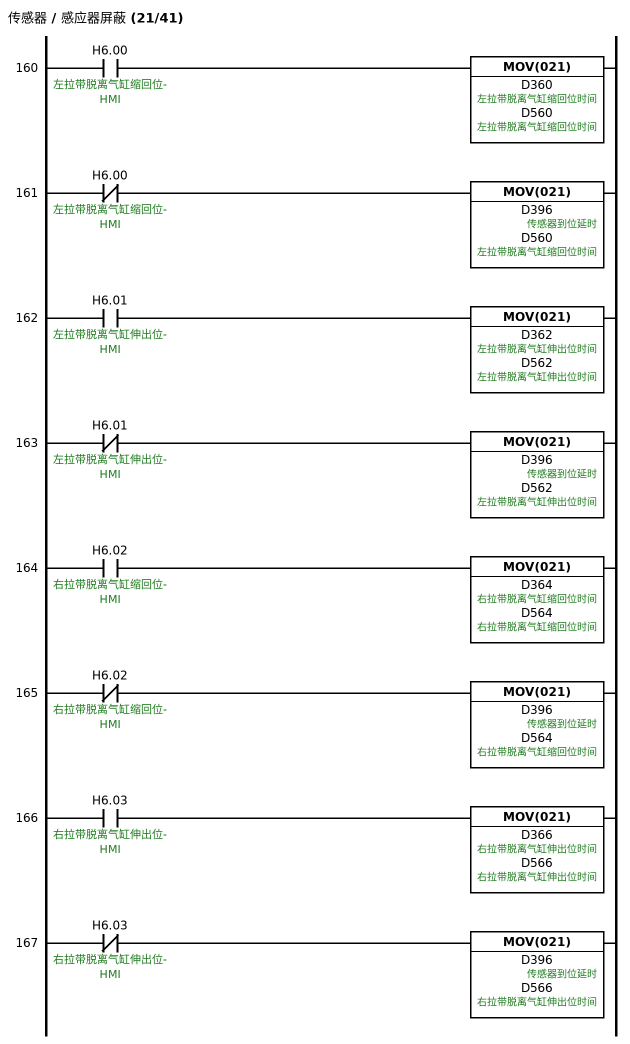
; [picture p41: 传感器 / 感应器屏蔽, rungs 160-167]
; rung 160
LD H6.00  ; 左拉带脱离气缸缩回位-HMI
MOV(021) D360 D560  ; 左拉带脱离气缸缩回位时间
; rung 161
LDNOT H6.00  ; 左拉带脱离气缸缩回位-HMI
MOV(021) D396 D560  ; 传感器到位延时, 左拉带脱离气缸缩回位时间
; rung 162
LD H6.01  ; 左拉带脱离气缸伸出位-HMI
MOV(021) D362 D562  ; 左拉带脱离气缸伸出位时间
; rung 163
LDNOT H6.01  ; 左拉带脱离气缸伸出位-HMI
MOV(021) D396 D562  ; 传感器到位延时, 左拉带脱离气缸伸出位时间
; rung 164
LD H6.02  ; 右拉带脱离气缸缩回位-HMI
MOV(021) D364 D564  ; 右拉带脱离气缸缩回位时间
; rung 165
LDNOT H6.02  ; 右拉带脱离气缸缩回位-HMI
MOV(021) D396 D564  ; 传感器到位延时, 右拉带脱离气缸缩回位时间
; rung 166
LD H6.03  ; 右拉带脱离气缸伸出位-HMI
MOV(021) D366 D566  ; 右拉带脱离气缸伸出位时间
; rung 167
LDNOT H6.03  ; 右拉带脱离气缸伸出位-HMI
MOV(021) D396 D566  ; 传感器到位延时, 右拉带脱离气缸伸出位时间

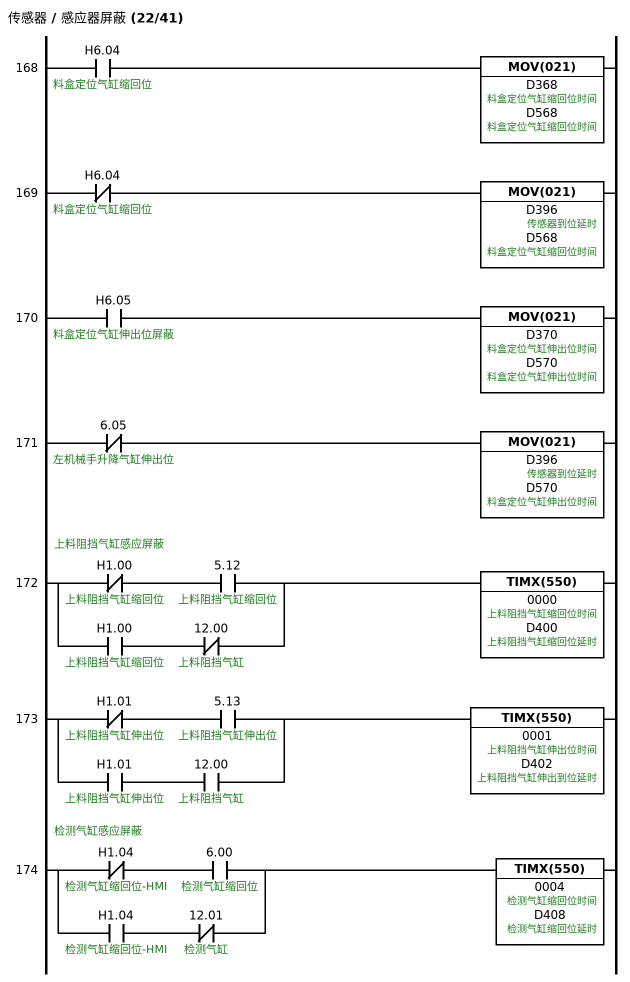
; rung 168
LD H6.04  ; 料盒定位气缸缩回位
MOV(021) D368 D568  ; 料盒定位气缸缩回位时间
; rung 169
LDNOT H6.04  ; 料盒定位气缸缩回位
MOV(021) D396 D568  ; 传感器到位延时, 料盒定位气缸缩回位时间
; rung 170
LD H6.05  ; 料盒定位气缸伸出位屏蔽
MOV(021) D370 D570  ; 料盒定位气缸伸出位时间
; rung 171
LDNOT 6.05  ; 左机械手升降气缸伸出位
MOV(021) D396 D570  ; 传感器到位延时, 料盒定位气缸伸出位时间
; rung 172: 上料阻挡气缸感应屏蔽
LDNOT H1.00  ; 上料阻挡气缸缩回位
AND 5.12  ; 上料阻挡气缸缩回位
LD H1.00  ; 上料阻挡气缸缩回位
ANDNOT 12.00  ; 上料阻挡气缸
ORLD
TIMX(550) 0000 D400  ; 上料阻挡气缸缩回位延时, 上料阻挡气缸缩回位时间
; rung 173
LDNOT H1.01  ; 上料阻挡气缸伸出位
AND 5.13  ; 上料阻挡气缸伸出位
LD H1.01  ; 上料阻挡气缸伸出位
AND 12.00  ; 上料阻挡气缸
ORLD
TIMX(550) 0001 D402  ; 上料阻挡气缸伸出到位延时, 上料阻挡气缸伸出位时间
; rung 174: 检测气缸感应屏蔽
LDNOT H1.04  ; 检测气缸缩回位-HMI
AND 6.00  ; 检测气缸缩回位
LD H1.04  ; 检测气缸缩回位-HMI
ANDNOT 12.01  ; 检测气缸
ORLD
TIMX(550) 0004 D408  ; 检测气缸缩回位延时, 检测气缸缩回位时间

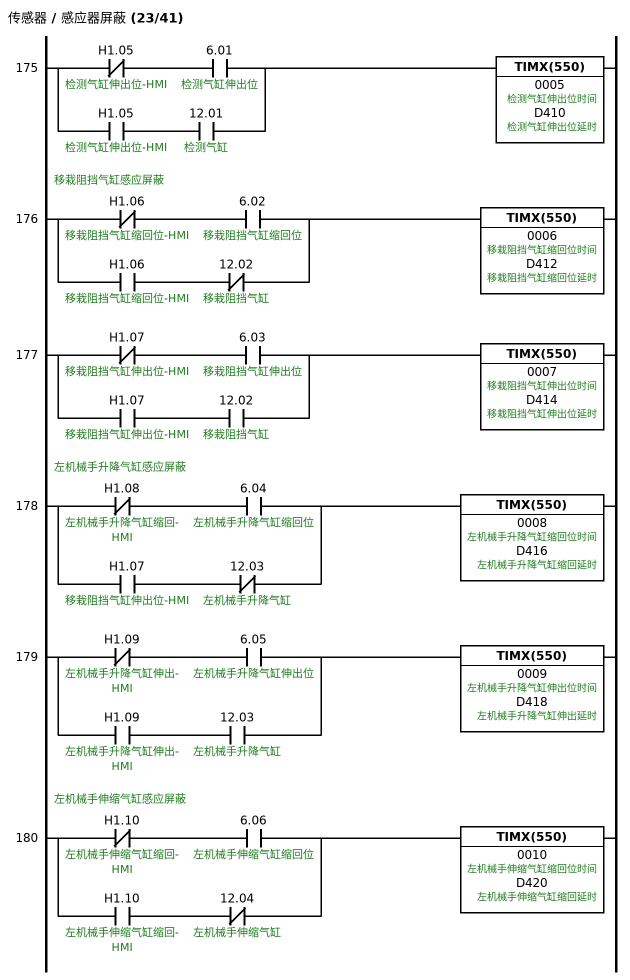
; rung 175
LDNOT H1.05  ; 检测气缸伸出位-HMI
AND 6.01  ; 检测气缸伸出位
LD H1.05  ; 检测气缸伸出位-HMI
AND 12.01  ; 检测气缸
ORLD
TIMX(550) 0005 D410  ; 检测气缸伸出位延时, 检测气缸伸出位时间
; rung 176: 移栽阻挡气缸感应屏蔽
LDNOT H1.06  ; 移栽阻挡气缸缩回位-HMI
AND 6.02  ; 移栽阻挡气缸缩回位
LD H1.06  ; 移栽阻挡气缸缩回位-HMI
ANDNOT 12.02  ; 移栽阻挡气缸
ORLD
TIMX(550) 0006 D412  ; 移栽阻挡气缸缩回位延时, 移栽阻挡气缸缩回位时间
; rung 177
LDNOT H1.07  ; 移栽阻挡气缸伸出位-HMI
AND 6.03  ; 移栽阻挡气缸伸出位
LD H1.07  ; 移栽阻挡气缸伸出位-HMI
AND 12.02  ; 移栽阻挡气缸
ORLD
TIMX(550) 0007 D414  ; 移栽阻挡气缸伸出位延时, 移栽阻挡气缸伸出位时间
; rung 178: 左机械手升降气缸感应屏蔽
LDNOT H1.08  ; 左机械手升降气缸缩回-HMI
AND 6.04  ; 左机械手升降气缸缩回位
LD H1.07  ; 移栽阻挡气缸伸出位-HMI
ANDNOT 12.03  ; 左机械手升降气缸
ORLD
TIMX(550) 0008 D416  ; 左机械手升降气缸缩回延时, 左机械手升降气缸缩回位时间
; rung 179
LDNOT H1.09  ; 左机械手升降气缸伸出-HMI
AND 6.05  ; 左机械手升降气缸伸出位
LD H1.09  ; 左机械手升降气缸伸出-HMI
AND 12.03  ; 左机械手升降气缸
ORLD
TIMX(550) 0009 D418  ; 左机械手升降气缸伸出延时, 左机械手升降气缸伸出位时间
; rung 180: 左机械手伸缩气缸感应屏蔽
LDNOT H1.10  ; 左机械手伸缩气缸缩回-HMI
AND 6.06  ; 左机械手伸缩气缸缩回位
LD H1.10  ; 左机械手伸缩气缸缩回-HMI
ANDNOT 12.04  ; 左机械手伸缩气缸
ORLD
TIMX(550) 0010 D420  ; 左机械手伸缩气缸缩回延时, 左机械手伸缩气缸缩回位时间

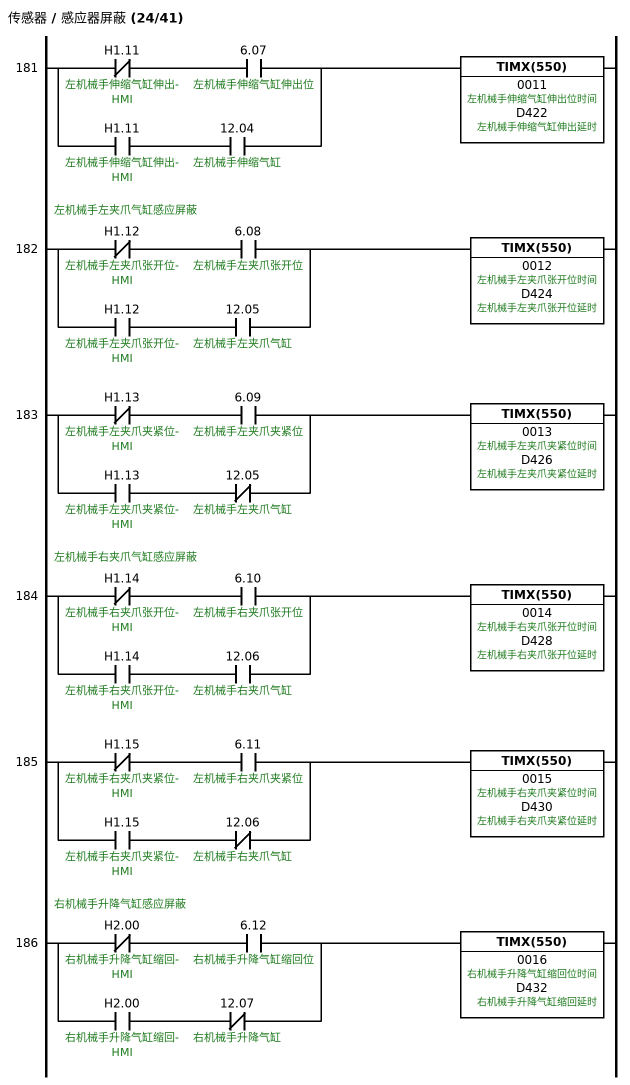
; rung 181
LDNOT H1.11  ; 左机械手伸缩气缸伸出-HMI
AND 6.07  ; 左机械手伸缩气缸伸出位
LD H1.11  ; 左机械手伸缩气缸伸出-HMI
AND 12.04  ; 左机械手伸缩气缸
ORLD
TIMX(550) 0011 D422  ; 左机械手伸缩气缸伸出延时, 左机械手伸缩气缸伸出位时间
; rung 182: 左机械手左夹爪气缸感应屏蔽
LDNOT H1.12  ; 左机械手左夹爪张开位-HMI
AND 6.08  ; 左机械手左夹爪张开位
LD H1.12  ; 左机械手左夹爪张开位-HMI
AND 12.05  ; 左机械手左夹爪气缸
ORLD
TIMX(550) 0012 D424  ; 左机械手左夹爪张开位延时, 左机械手左夹爪张开位时间
; rung 183
LDNOT H1.13  ; 左机械手左夹爪夹紧位-HMI
AND 6.09  ; 左机械手左夹爪夹紧位
LD H1.13  ; 左机械手左夹爪夹紧位-HMI
ANDNOT 12.05  ; 左机械手左夹爪气缸
ORLD
TIMX(550) 0013 D426  ; 左机械手左夹爪夹紧位延时, 左机械手左夹爪夹紧位时间
; rung 184: 左机械手右夹爪气缸感应屏蔽
LDNOT H1.14  ; 左机械手右夹爪张开位-HMI
AND 6.10  ; 左机械手右夹爪张开位
LD H1.14  ; 左机械手右夹爪张开位-HMI
AND 12.06  ; 左机械手右夹爪气缸
ORLD
TIMX(550) 0014 D428  ; 左机械手右夹爪张开位延时, 左机械手右夹爪张开位时间
; rung 185
LDNOT H1.15  ; 左机械手右夹爪夹紧位-HMI
AND 6.11  ; 左机械手右夹爪夹紧位
LD H1.15  ; 左机械手右夹爪夹紧位-HMI
ANDNOT 12.06  ; 左机械手右夹爪气缸
ORLD
TIMX(550) 0015 D430  ; 左机械手右夹爪夹紧位延时, 左机械手右夹爪夹紧位时间
; rung 186: 右机械手升降气缸感应屏蔽
LDNOT H2.00  ; 右机械手升降气缸缩回-HMI
AND 6.12  ; 右机械手升降气缸缩回位
LD H2.00  ; 右机械手升降气缸缩回-HMI
ANDNOT 12.07  ; 右机械手升降气缸
ORLD
TIMX(550) 0016 D432  ; 右机械手升降气缸缩回延时, 右机械手升降气缸缩回位时间

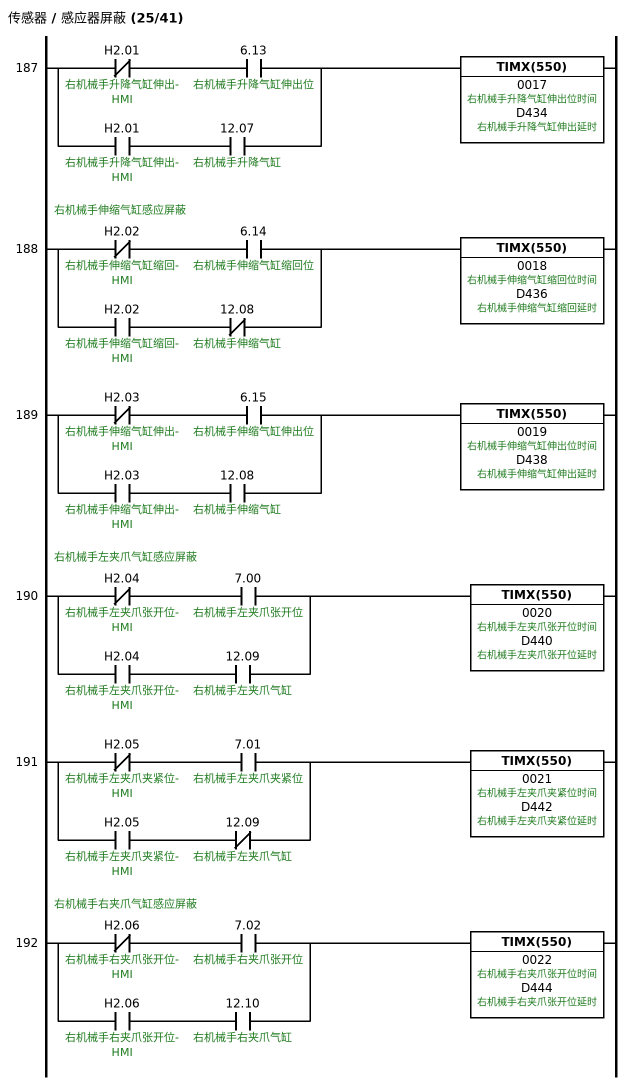
; rung 187
LDNOT H2.01  ; 右机械手升降气缸伸出-HMI
AND 6.13  ; 右机械手升降气缸伸出位
LD H2.01  ; 右机械手升降气缸伸出-HMI
AND 12.07  ; 右机械手升降气缸
ORLD
TIMX(550) 0017 D434  ; 右机械手升降气缸伸出延时, 右机械手升降气缸伸出位时间
; rung 188: 右机械手伸缩气缸感应屏蔽
LDNOT H2.02  ; 右机械手伸缩气缸缩回-HMI
AND 6.14  ; 右机械手伸缩气缸缩回位
LD H2.02  ; 右机械手伸缩气缸缩回-HMI
ANDNOT 12.08  ; 右机械手伸缩气缸
ORLD
TIMX(550) 0018 D436  ; 右机械手伸缩气缸缩回延时, 右机械手伸缩气缸缩回位时间
; rung 189
LDNOT H2.03  ; 右机械手伸缩气缸伸出-HMI
AND 6.15  ; 右机械手伸缩气缸伸出位
LD H2.03  ; 右机械手伸缩气缸伸出-HMI
AND 12.08  ; 右机械手伸缩气缸
ORLD
TIMX(550) 0019 D438  ; 右机械手伸缩气缸伸出延时, 右机械手伸缩气缸伸出位时间
; rung 190: 右机械手左夹爪气缸感应屏蔽
LDNOT H2.04  ; 右机械手左夹爪张开位-HMI
AND 7.00  ; 右机械手左夹爪张开位
LD H2.04  ; 右机械手左夹爪张开位-HMI
AND 12.09  ; 右机械手左夹爪气缸
ORLD
TIMX(550) 0020 D440  ; 右机械手左夹爪张开位延时, 右机械手左夹爪张开位时间
; rung 191
LDNOT H2.05  ; 右机械手左夹爪夹紧位-HMI
AND 7.01  ; 右机械手左夹爪夹紧位
LD H2.05  ; 右机械手左夹爪夹紧位-HMI
ANDNOT 12.09  ; 右机械手左夹爪气缸
ORLD
TIMX(550) 0021 D442  ; 右机械手左夹爪夹紧位延时, 右机械手左夹爪夹紧位时间
; rung 192: 右机械手右夹爪气缸感应屏蔽
LDNOT H2.06  ; 右机械手右夹爪张开位-HMI
AND 7.02  ; 右机械手右夹爪张开位
LD H2.06  ; 右机械手右夹爪张开位-HMI
AND 12.10  ; 右机械手右夹爪气缸
ORLD
TIMX(550) 0022 D444  ; 右机械手右夹爪张开位延时, 右机械手右夹爪张开位时间

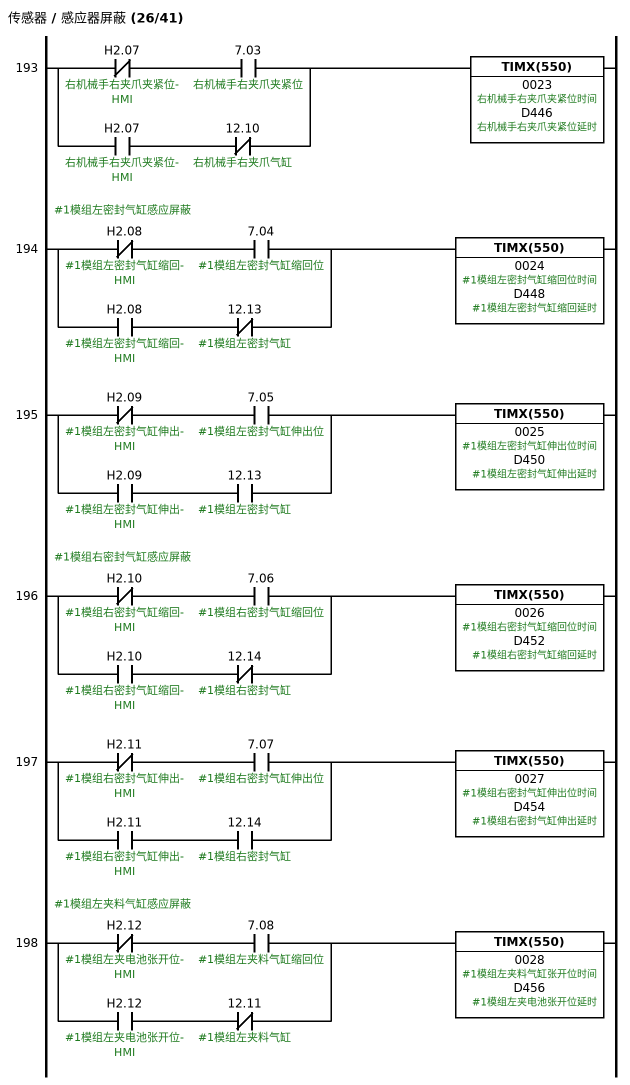
; rung 193
LDNOT H2.07  ; 右机械手右夹爪夹紧位-HMI
AND 7.03  ; 右机械手右夹爪夹紧位
LD H2.07  ; 右机械手右夹爪夹紧位-HMI
ANDNOT 12.10  ; 右机械手右夹爪气缸
ORLD
TIMX(550) 0023 D446  ; 右机械手右夹爪夹紧位延时, 右机械手右夹爪夹紧位时间
; rung 194: #1模组左密封气缸感应屏蔽
LDNOT H2.08  ; #1模组左密封气缸缩回-HMI
AND 7.04  ; #1模组左密封气缸缩回位
LD H2.08  ; #1模组左密封气缸缩回-HMI
ANDNOT 12.13  ; #1模组左密封气缸
ORLD
TIMX(550) 0024 D448  ; #1模组左密封气缸缩回延时, #1模组左密封气缸缩回位时间
; rung 195
LDNOT H2.09  ; #1模组左密封气缸伸出-HMI
AND 7.05  ; #1模组左密封气缸伸出位
LD H2.09  ; #1模组左密封气缸伸出-HMI
AND 12.13  ; #1模组左密封气缸
ORLD
TIMX(550) 0025 D450  ; #1模组左密封气缸伸出延时, #1模组左密封气缸伸出位时间
; rung 196: #1模组右密封气缸感应屏蔽
LDNOT H2.10  ; #1模组右密封气缸缩回-HMI
AND 7.06  ; #1模组右密封气缸缩回位
LD H2.10  ; #1模组右密封气缸缩回-HMI
ANDNOT 12.14  ; #1模组右密封气缸
ORLD
TIMX(550) 0026 D452  ; #1模组右密封气缸缩回延时, #1模组右密封气缸缩回位时间
; rung 197
LDNOT H2.11  ; #1模组右密封气缸伸出-HMI
AND 7.07  ; #1模组右密封气缸伸出位
LD H2.11  ; #1模组右密封气缸伸出-HMI
AND 12.14  ; #1模组右密封气缸
ORLD
TIMX(550) 0027 D454  ; #1模组右密封气缸伸出延时, #1模组右密封气缸伸出位时间
; rung 198: #1模组左夹料气缸感应屏蔽
LDNOT H2.12  ; #1模组左夹电池张开位-HMI
AND 7.08  ; #1模组左夹料气缸缩回位
LD H2.12  ; #1模组左夹电池张开位-HMI
ANDNOT 12.11  ; #1模组左夹料气缸
ORLD
TIMX(550) 0028 D456  ; #1模组左夹电池张开位延时, #1模组左夹料气缸张开位时间

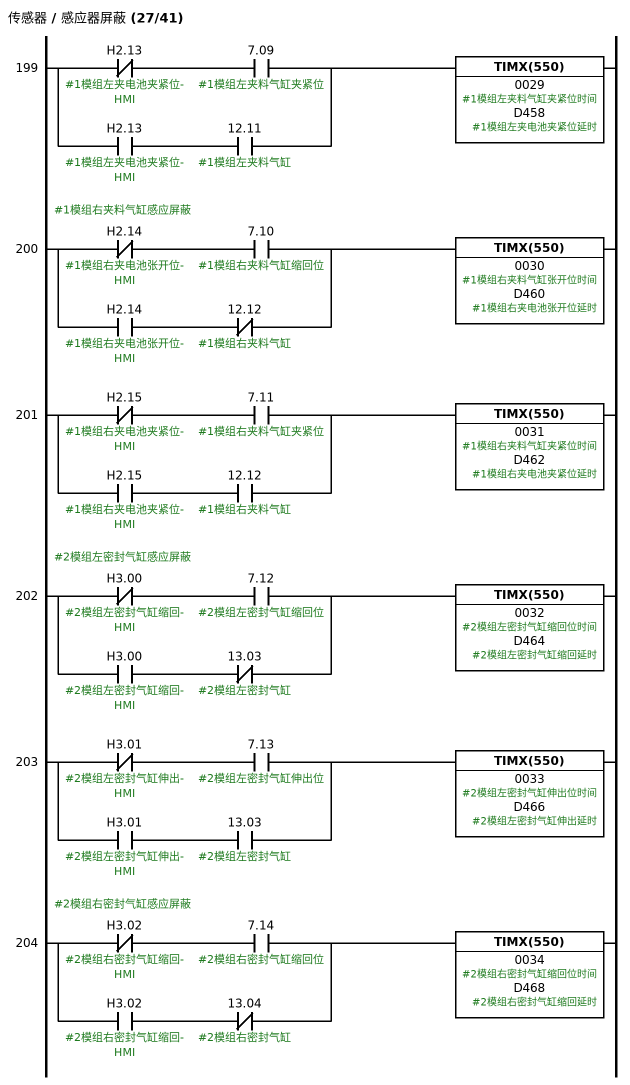
; rung 199
LDNOT H2.13  ; #1模组左夹电池夹紧位-HMI
AND 7.09  ; #1模组左夹料气缸夹紧位
LD H2.13  ; #1模组左夹电池夹紧位-HMI
AND 12.11  ; #1模组左夹料气缸
ORLD
TIMX(550) 0029 D458  ; #1模组左夹电池夹紧位延时, #1模组左夹料气缸夹紧位时间
; rung 200: #1模组右夹料气缸感应屏蔽
LDNOT H2.14  ; #1模组右夹电池张开位-HMI
AND 7.10  ; #1模组右夹料气缸缩回位
LD H2.14  ; #1模组右夹电池张开位-HMI
ANDNOT 12.12  ; #1模组右夹料气缸
ORLD
TIMX(550) 0030 D460  ; #1模组右夹电池张开位延时, #1模组右夹料气缸张开位时间
; rung 201
LDNOT H2.15  ; #1模组右夹电池夹紧位-HMI
AND 7.11  ; #1模组右夹料气缸夹紧位
LD H2.15  ; #1模组右夹电池夹紧位-HMI
AND 12.12  ; #1模组右夹料气缸
ORLD
TIMX(550) 0031 D462  ; #1模组右夹电池夹紧位延时, #1模组右夹料气缸夹紧位时间
; rung 202: #2模组左密封气缸感应屏蔽
LDNOT H3.00  ; #2模组左密封气缸缩回-HMI
AND 7.12  ; #2模组左密封气缸缩回位
LD H3.00  ; #2模组左密封气缸缩回-HMI
ANDNOT 13.03  ; #2模组左密封气缸
ORLD
TIMX(550) 0032 D464  ; #2模组左密封气缸缩回延时, #2模组左密封气缸缩回位时间
; rung 203
LDNOT H3.01  ; #2模组左密封气缸伸出-HMI
AND 7.13  ; #2模组左密封气缸伸出位
LD H3.01  ; #2模组左密封气缸伸出-HMI
AND 13.03  ; #2模组左密封气缸
ORLD
TIMX(550) 0033 D466  ; #2模组左密封气缸伸出延时, #2模组左密封气缸伸出位时间
; rung 204: #2模组右密封气缸感应屏蔽
LDNOT H3.02  ; #2模组右密封气缸缩回-HMI
AND 7.14  ; #2模组右密封气缸缩回位
LD H3.02  ; #2模组右密封气缸缩回-HMI
ANDNOT 13.04  ; #2模组右密封气缸
ORLD
TIMX(550) 0034 D468  ; #2模组右密封气缸缩回延时, #2模组右密封气缸缩回位时间

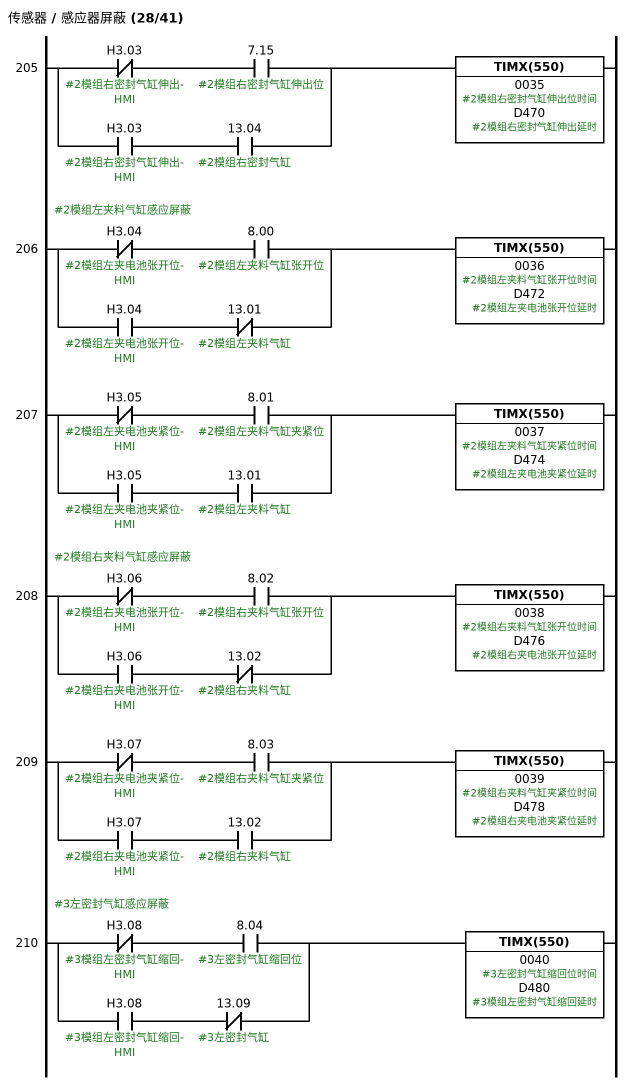
; rung 205
LDNOT H3.03  ; #2模组右密封气缸伸出-HMI
AND 7.15  ; #2模组右密封气缸伸出位
LD H3.03  ; #2模组右密封气缸伸出-HMI
AND 13.04  ; #2模组右密封气缸
ORLD
TIMX(550) 0035 D470  ; #2模组右密封气缸伸出延时, #2模组右密封气缸伸出位时间
; rung 206: #2模组左夹料气缸感应屏蔽
LDNOT H3.04  ; #2模组左夹电池张开位-HMI
AND 8.00  ; #2模组左夹料气缸张开位
LD H3.04  ; #2模组左夹电池张开位-HMI
ANDNOT 13.01  ; #2模组左夹料气缸
ORLD
TIMX(550) 0036 D472  ; #2模组左夹电池张开位延时, #2模组左夹料气缸张开位时间
; rung 207
LDNOT H3.05  ; #2模组左夹电池夹紧位-HMI
AND 8.01  ; #2模组左夹料气缸夹紧位
LD H3.05  ; #2模组左夹电池夹紧位-HMI
AND 13.01  ; #2模组左夹料气缸
ORLD
TIMX(550) 0037 D474  ; #2模组左夹电池夹紧位延时, #2模组左夹料气缸夹紧位时间
; rung 208: #2模组右夹料气缸感应屏蔽
LDNOT H3.06  ; #2模组右夹电池张开位-HMI
AND 8.02  ; #2模组右夹料气缸张开位
LD H3.06  ; #2模组右夹电池张开位-HMI
ANDNOT 13.02  ; #2模组右夹料气缸
ORLD
TIMX(550) 0038 D476  ; #2模组右夹电池张开位延时, #2模组右夹料气缸张开位时间
; rung 209
LDNOT H3.07  ; #2模组右夹电池夹紧位-HMI
AND 8.03  ; #2模组右夹料气缸夹紧位
LD H3.07  ; #2模组右夹电池夹紧位-HMI
AND 13.02  ; #2模组右夹料气缸
ORLD
TIMX(550) 0039 D478  ; #2模组右夹电池夹紧位延时, #2模组右夹料气缸夹紧位时间
; rung 210: #3左密封气缸感应屏蔽
LDNOT H3.08  ; #3模组左密封气缸缩回-HMI
AND 8.04  ; #3左密封气缸缩回位
LD H3.08  ; #3模组左密封气缸缩回-HMI
ANDNOT 13.09  ; #3左密封气缸
ORLD
TIMX(550) 0040 D480  ; #3模组左密封气缸缩回延时, #3左密封气缸缩回位时间

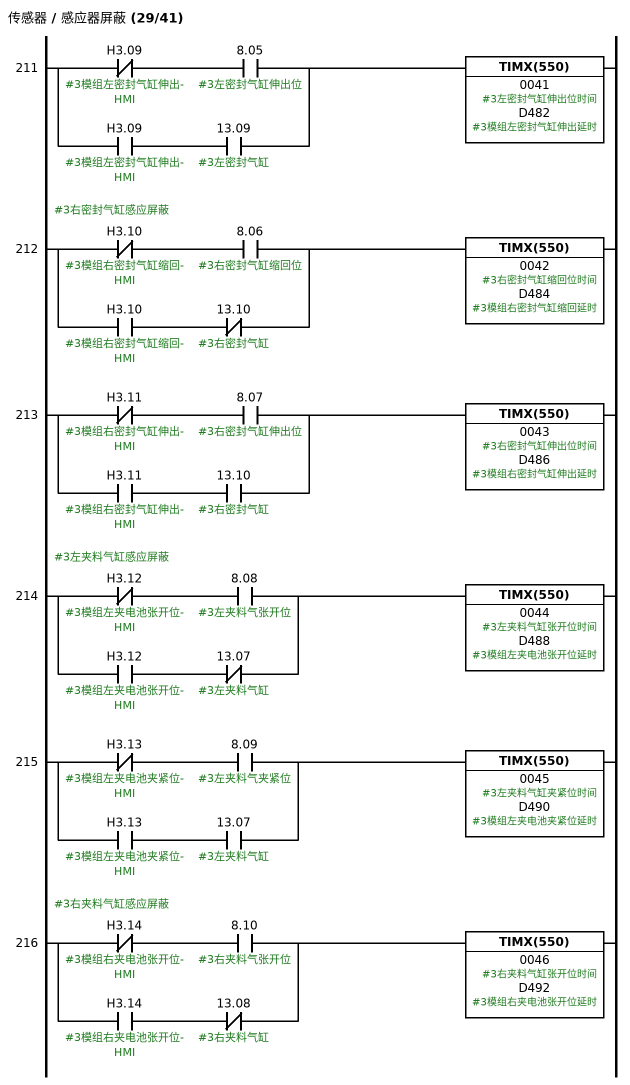
; rung 211
LDNOT H3.09  ; #3模组左密封气缸伸出-HMI
AND 8.05  ; #3左密封气缸伸出位
LD H3.09  ; #3模组左密封气缸伸出-HMI
AND 13.09  ; #3左密封气缸
ORLD
TIMX(550) 0041 D482  ; #3模组左密封气缸伸出延时, #3左密封气缸伸出位时间
; rung 212: #3右密封气缸感应屏蔽
LDNOT H3.10  ; #3模组右密封气缸缩回-HMI
AND 8.06  ; #3右密封气缸缩回位
LD H3.10  ; #3模组右密封气缸缩回-HMI
ANDNOT 13.10  ; #3右密封气缸
ORLD
TIMX(550) 0042 D484  ; #3模组右密封气缸缩回延时, #3右密封气缸缩回位时间
; rung 213
LDNOT H3.11  ; #3模组右密封气缸伸出-HMI
AND 8.07  ; #3右密封气缸伸出位
LD H3.11  ; #3模组右密封气缸伸出-HMI
AND 13.10  ; #3右密封气缸
ORLD
TIMX(550) 0043 D486  ; #3模组右密封气缸伸出延时, #3右密封气缸伸出位时间
; rung 214: #3左夹料气缸感应屏蔽
LDNOT H3.12  ; #3模组左夹电池张开位-HMI
AND 8.08  ; #3左夹料气张开位
LD H3.12  ; #3模组左夹电池张开位-HMI
ANDNOT 13.07  ; #3左夹料气缸
ORLD
TIMX(550) 0044 D488  ; #3模组左夹电池张开位延时, #3左夹料气缸张开位时间
; rung 215
LDNOT H3.13  ; #3模组左夹电池夹紧位-HMI
AND 8.09  ; #3左夹料气夹紧位
LD H3.13  ; #3模组左夹电池夹紧位-HMI
AND 13.07  ; #3左夹料气缸
ORLD
TIMX(550) 0045 D490  ; #3模组左夹电池夹紧位延时, #3左夹料气缸夹紧位时间
; rung 216: #3右夹料气缸感应屏蔽
LDNOT H3.14  ; #3模组右夹电池张开位-HMI
AND 8.10  ; #3右夹料气张开位
LD H3.14  ; #3模组右夹电池张开位-HMI
ANDNOT 13.08  ; #3右夹料气缸
ORLD
TIMX(550) 0046 D492  ; #3模组右夹电池张开位延时, #3右夹料气缸张开位时间

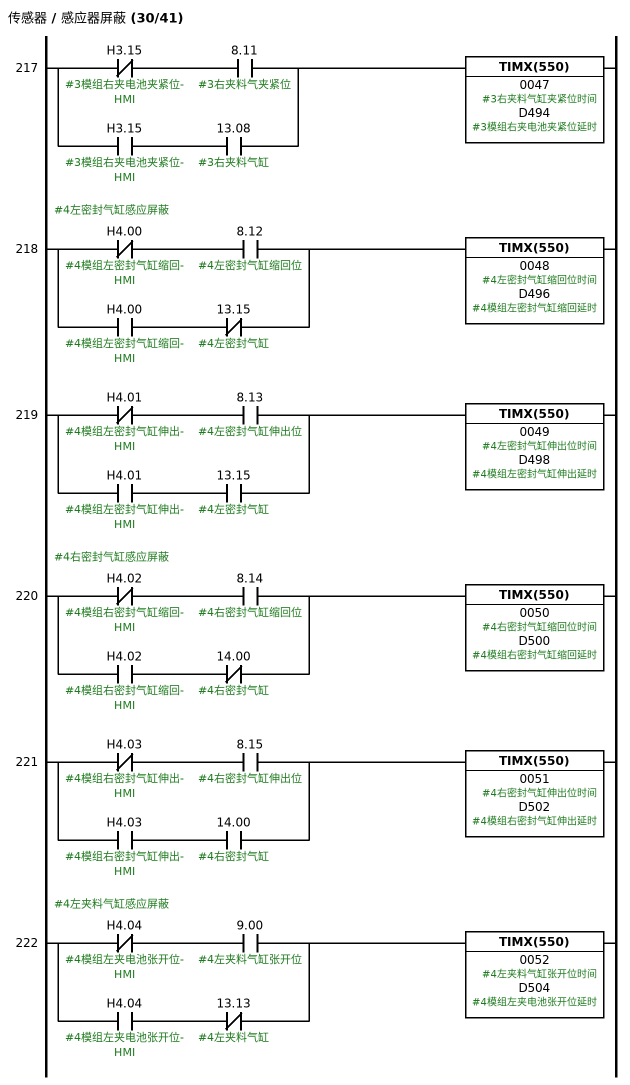
; rung 217
LDNOT H3.15  ; #3模组右夹电池夹紧位-HMI
AND 8.11  ; #3右夹料气夹紧位
LD H3.15  ; #3模组右夹电池夹紧位-HMI
AND 13.08  ; #3右夹料气缸
ORLD
TIMX(550) 0047 D494  ; #3模组右夹电池夹紧位延时, #3右夹料气缸夹紧位时间
; rung 218: #4左密封气缸感应屏蔽
LDNOT H4.00  ; #4模组左密封气缸缩回-HMI
AND 8.12  ; #4左密封气缸缩回位
LD H4.00  ; #4模组左密封气缸缩回-HMI
ANDNOT 13.15  ; #4左密封气缸
ORLD
TIMX(550) 0048 D496  ; #4模组左密封气缸缩回延时, #4左密封气缸缩回位时间
; rung 219
LDNOT H4.01  ; #4模组左密封气缸伸出-HMI
AND 8.13  ; #4左密封气缸伸出位
LD H4.01  ; #4模组左密封气缸伸出-HMI
AND 13.15  ; #4左密封气缸
ORLD
TIMX(550) 0049 D498  ; #4模组左密封气缸伸出延时, #4左密封气缸伸出位时间
; rung 220: #4右密封气缸感应屏蔽
LDNOT H4.02  ; #4模组右密封气缸缩回-HMI
AND 8.14  ; #4右密封气缸缩回位
LD H4.02  ; #4模组右密封气缸缩回-HMI
ANDNOT 14.00  ; #4右密封气缸
ORLD
TIMX(550) 0050 D500  ; #4模组右密封气缸缩回延时, #4右密封气缸缩回位时间
; rung 221
LDNOT H4.03  ; #4模组右密封气缸伸出-HMI
AND 8.15  ; #4右密封气缸伸出位
LD H4.03  ; #4模组右密封气缸伸出-HMI
AND 14.00  ; #4右密封气缸
ORLD
TIMX(550) 0051 D502  ; #4模组右密封气缸伸出延时, #4右密封气缸伸出位时间
; rung 222: #4左夹料气缸感应屏蔽
LDNOT H4.04  ; #4模组左夹电池张开位-HMI
AND 9.00  ; #4左夹料气缸张开位
LD H4.04  ; #4模组左夹电池张开位-HMI
ANDNOT 13.13  ; #4左夹料气缸
ORLD
TIMX(550) 0052 D504  ; #4模组左夹电池张开位延时, #4左夹料气缸张开位时间

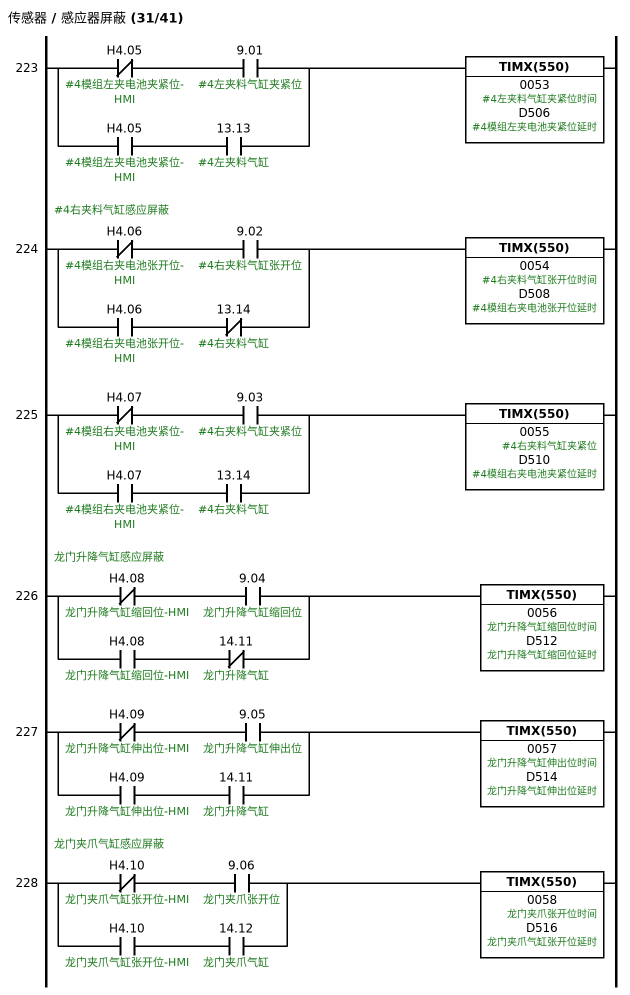
; rung 223
LDNOT H4.05  ; #4模组左夹电池夹紧位-HMI
AND 9.01  ; #4左夹料气缸夹紧位
LD H4.05  ; #4模组左夹电池夹紧位-HMI
AND 13.13  ; #4左夹料气缸
ORLD
TIMX(550) 0053 D506  ; #4模组左夹电池夹紧位延时, #4左夹料气缸夹紧位时间
; rung 224: #4右夹料气缸感应屏蔽
LDNOT H4.06  ; #4模组右夹电池张开位-HMI
AND 9.02  ; #4右夹料气缸张开位
LD H4.06  ; #4模组右夹电池张开位-HMI
ANDNOT 13.14  ; #4右夹料气缸
ORLD
TIMX(550) 0054 D508  ; #4模组右夹电池张开位延时, #4右夹料气缸张开位时间
; rung 225
LDNOT H4.07  ; #4模组右夹电池夹紧位-HMI
AND 9.03  ; #4右夹料气缸夹紧位
LD H4.07  ; #4模组右夹电池夹紧位-HMI
AND 13.14  ; #4右夹料气缸
ORLD
TIMX(550) 0055 D510  ; #4模组右夹电池夹紧位延时, #4右夹料气缸夹紧位
; rung 226: 龙门升降气缸感应屏蔽
LDNOT H4.08  ; 龙门升降气缸缩回位-HMI
AND 9.04  ; 龙门升降气缸缩回位
LD H4.08  ; 龙门升降气缸缩回位-HMI
ANDNOT 14.11  ; 龙门升降气缸
ORLD
TIMX(550) 0056 D512  ; 龙门升降气缸缩回位延时, 龙门升降气缸缩回位时间
; rung 227
LDNOT H4.09  ; 龙门升降气缸伸出位-HMI
AND 9.05  ; 龙门升降气缸伸出位
LD H4.09  ; 龙门升降气缸伸出位-HMI
AND 14.11  ; 龙门升降气缸
ORLD
TIMX(550) 0057 D514  ; 龙门升降气缸伸出位延时, 龙门升降气缸伸出位时间
; rung 228: 龙门夹爪气缸感应屏蔽
LDNOT H4.10  ; 龙门夹爪气缸张开位-HMI
AND 9.06  ; 龙门夹爪张开位
LD H4.10  ; 龙门夹爪气缸张开位-HMI
AND 14.12  ; 龙门夹爪气缸
ORLD
TIMX(550) 0058 D516  ; 龙门夹爪气缸张开位延时, 龙门夹爪张开位时间

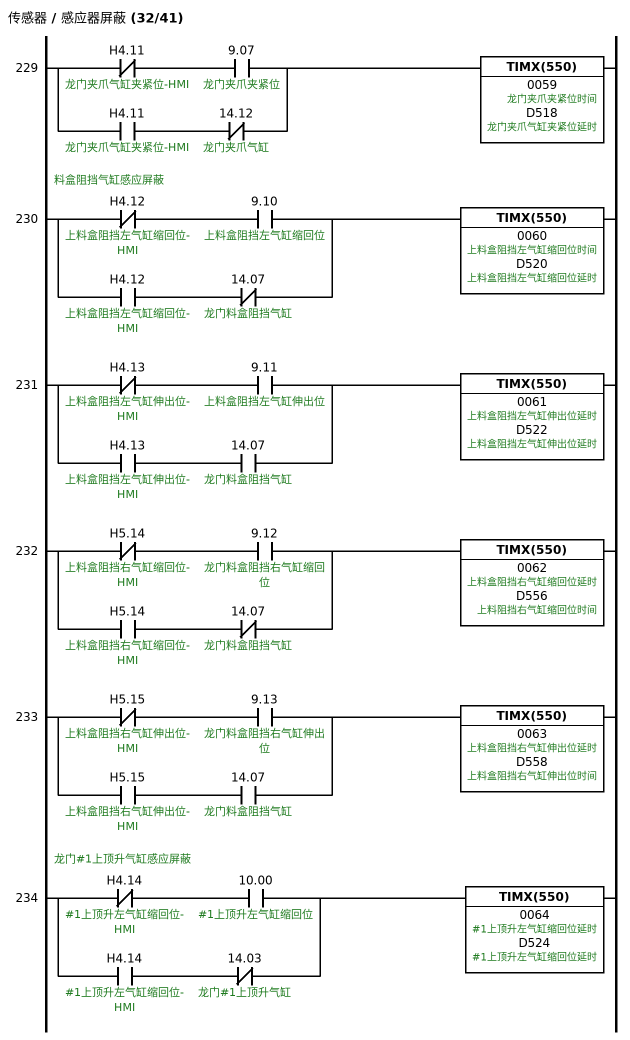
; rung 229
LDNOT H4.11  ; 龙门夹爪气缸夹紧位-HMI
AND 9.07  ; 龙门夹爪夹紧位
LD H4.11  ; 龙门夹爪气缸夹紧位-HMI
ANDNOT 14.12  ; 龙门夹爪气缸
ORLD
TIMX(550) 0059 D518  ; 龙门夹爪气缸夹紧位延时, 龙门夹爪夹紧位时间
; rung 230: 料盒阻挡气缸感应屏蔽
LDNOT H4.12  ; 上料盒阻挡左气缸缩回位-HMI
AND 9.10  ; 上料盒阻挡左气缸缩回位
LD H4.12  ; 上料盒阻挡左气缸缩回位-HMI
ANDNOT 14.07  ; 龙门料盒阻挡气缸
ORLD
TIMX(550) 0060 D520  ; 上料盒阻挡左气缸缩回位延时, 上料盒阻挡左气缸缩回位时间
; rung 231
LDNOT H4.13  ; 上料盒阻挡左气缸伸出位-HMI
AND 9.11  ; 上料盒阻挡左气缸伸出位
LD H4.13  ; 上料盒阻挡左气缸伸出位-HMI
AND 14.07  ; 龙门料盒阻挡气缸
ORLD
TIMX(550) 0061 D522  ; 上料盒阻挡左气缸伸出位延时
; rung 232
LDNOT H5.14  ; 上料盒阻挡右气缸缩回位-HMI
AND 9.12  ; 龙门料盒阻挡右气缸缩回位
LD H5.14  ; 上料盒阻挡右气缸缩回位-HMI
ANDNOT 14.07  ; 龙门料盒阻挡气缸
ORLD
TIMX(550) 0062 D556  ; 上料阻挡右气缸缩回位时间, 上料盒阻挡右气缸缩回位延时
; rung 233
LDNOT H5.15  ; 上料盒阻挡右气缸伸出位-HMI
AND 9.13  ; 龙门料盒阻挡右气缸伸出位
LD H5.15  ; 上料盒阻挡右气缸伸出位-HMI
AND 14.07  ; 龙门料盒阻挡气缸
ORLD
TIMX(550) 0063 D558  ; 上料盒阻挡右气缸伸出位时间, 上料盒阻挡右气缸伸出位延时
; rung 234: 龙门#1上顶升气缸感应屏蔽
LDNOT H4.14  ; #1上顶升左气缸缩回位-HMI
AND 10.00  ; #1上顶升左气缸缩回位
LD H4.14  ; #1上顶升左气缸缩回位-HMI
ANDNOT 14.03  ; 龙门#1上顶升气缸
ORLD
TIMX(550) 0064 D524  ; #1上顶升左气缸缩回位延时

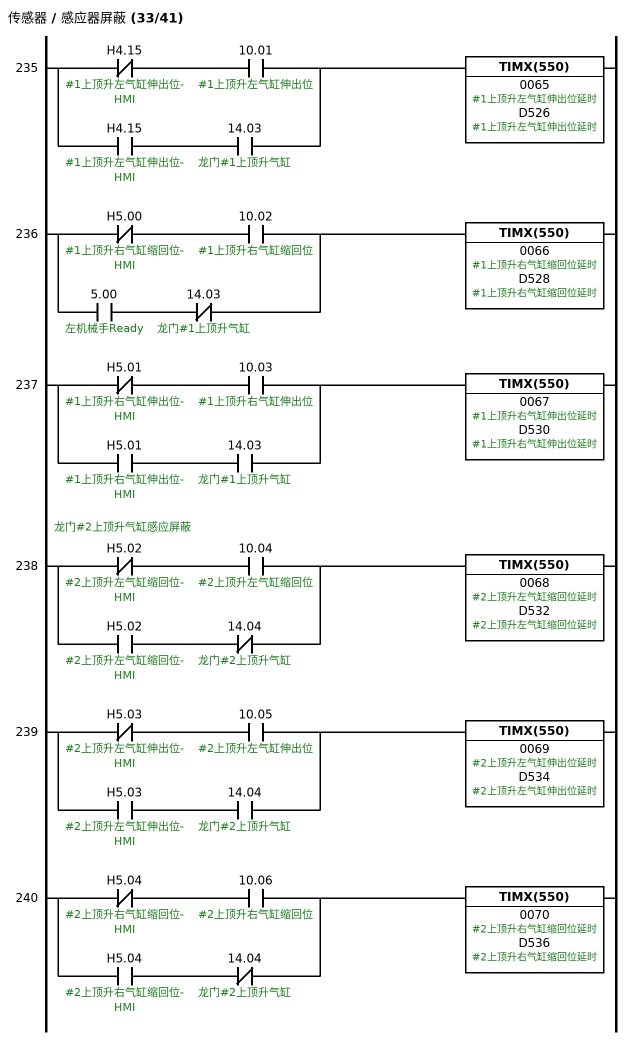
; rung 235
LDNOT H4.15  ; #1上顶升左气缸伸出位-HMI
AND 10.01  ; #1上顶升左气缸伸出位
LD H4.15  ; #1上顶升左气缸伸出位-HMI
AND 14.03  ; 龙门#1上顶升气缸
ORLD
TIMX(550) 0065 D526  ; #1上顶升左气缸伸出位延时
; rung 236
LDNOT H5.00  ; #1上顶升右气缸缩回位-HMI
AND 10.02  ; #1上顶升右气缸缩回位
LD 5.00  ; 左机械手Ready
ANDNOT 14.03  ; 龙门#1上顶升气缸
ORLD
TIMX(550) 0066 D528  ; #1上顶升右气缸缩回位延时
; rung 237
LDNOT H5.01  ; #1上顶升右气缸伸出位-HMI
AND 10.03  ; #1上顶升右气缸伸出位
LD H5.01  ; #1上顶升右气缸伸出位-HMI
AND 14.03  ; 龙门#1上顶升气缸
ORLD
TIMX(550) 0067 D530  ; #1上顶升右气缸伸出位延时
; rung 238: 龙门#2上顶升气缸感应屏蔽
LDNOT H5.02  ; #2上顶升左气缸缩回位-HMI
AND 10.04  ; #2上顶升左气缸缩回位
LD H5.02  ; #2上顶升左气缸缩回位-HMI
ANDNOT 14.04  ; 龙门#2上顶升气缸
ORLD
TIMX(550) 0068 D532  ; #2上顶升左气缸缩回位延时
; rung 239
LDNOT H5.03  ; #2上顶升左气缸伸出位-HMI
AND 10.05  ; #2上顶升左气缸伸出位
LD H5.03  ; #2上顶升左气缸伸出位-HMI
AND 14.04  ; 龙门#2上顶升气缸
ORLD
TIMX(550) 0069 D534  ; #2上顶升左气缸伸出位延时
; rung 240
LDNOT H5.04  ; #2上顶升右气缸缩回位-HMI
AND 10.06  ; #2上顶升右气缸缩回位
LD H5.04  ; #2上顶升右气缸缩回位-HMI
ANDNOT 14.04  ; 龙门#2上顶升气缸
ORLD
TIMX(550) 0070 D536  ; #2上顶升右气缸缩回位延时

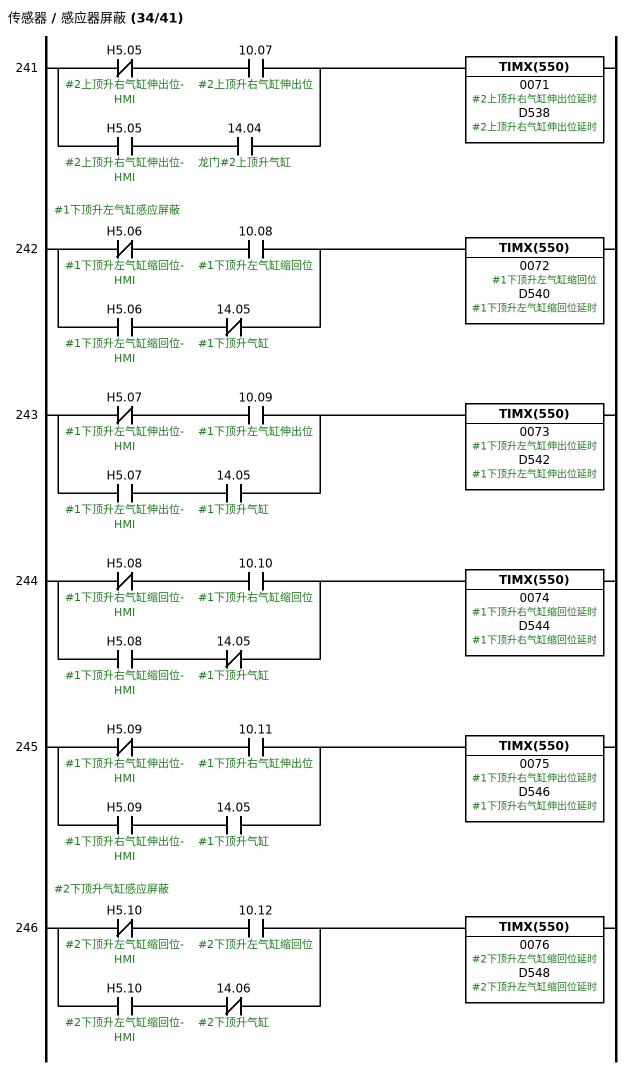
; rung 241
LDNOT H5.05  ; #2上顶升右气缸伸出位-HMI
AND 10.07  ; #2上顶升右气缸伸出位
LD H5.05  ; #2上顶升右气缸伸出位-HMI
AND 14.04  ; 龙门#2上顶升气缸
ORLD
TIMX(550) 0071 D538  ; #2上顶升右气缸伸出位延时
; rung 242: #1下顶升左气缸感应屏蔽
LDNOT H5.06  ; #1下顶升左气缸缩回位-HMI
AND 10.08  ; #1下顶升左气缸缩回位
LD H5.06  ; #1下顶升左气缸缩回位-HMI
ANDNOT 14.05  ; #1下顶升气缸
ORLD
TIMX(550) 0072 D540  ; #1下顶升左气缸缩回位延时, #1下顶升左气缸缩回位
; rung 243
LDNOT H5.07  ; #1下顶升左气缸伸出位-HMI
AND 10.09  ; #1下顶升左气缸伸出位
LD H5.07  ; #1下顶升左气缸伸出位-HMI
AND 14.05  ; #1下顶升气缸
ORLD
TIMX(550) 0073 D542  ; #1下顶升左气缸伸出位延时
; rung 244
LDNOT H5.08  ; #1下顶升右气缸缩回位-HMI
AND 10.10  ; #1下顶升右气缸缩回位
LD H5.08  ; #1下顶升右气缸缩回位-HMI
ANDNOT 14.05  ; #1下顶升气缸
ORLD
TIMX(550) 0074 D544  ; #1下顶升右气缸缩回位延时
; rung 245
LDNOT H5.09  ; #1下顶升右气缸伸出位-HMI
AND 10.11  ; #1下顶升右气缸伸出位
LD H5.09  ; #1下顶升右气缸伸出位-HMI
AND 14.05  ; #1下顶升气缸
ORLD
TIMX(550) 0075 D546  ; #1下顶升右气缸伸出位延时
; rung 246: #2下顶升气缸感应屏蔽
LDNOT H5.10  ; #2下顶升左气缸缩回位-HMI
AND 10.12  ; #2下顶升左气缸缩回位
LD H5.10  ; #2下顶升左气缸缩回位-HMI
ANDNOT 14.06  ; #2下顶升气缸
ORLD
TIMX(550) 0076 D548  ; #2下顶升左气缸缩回位延时

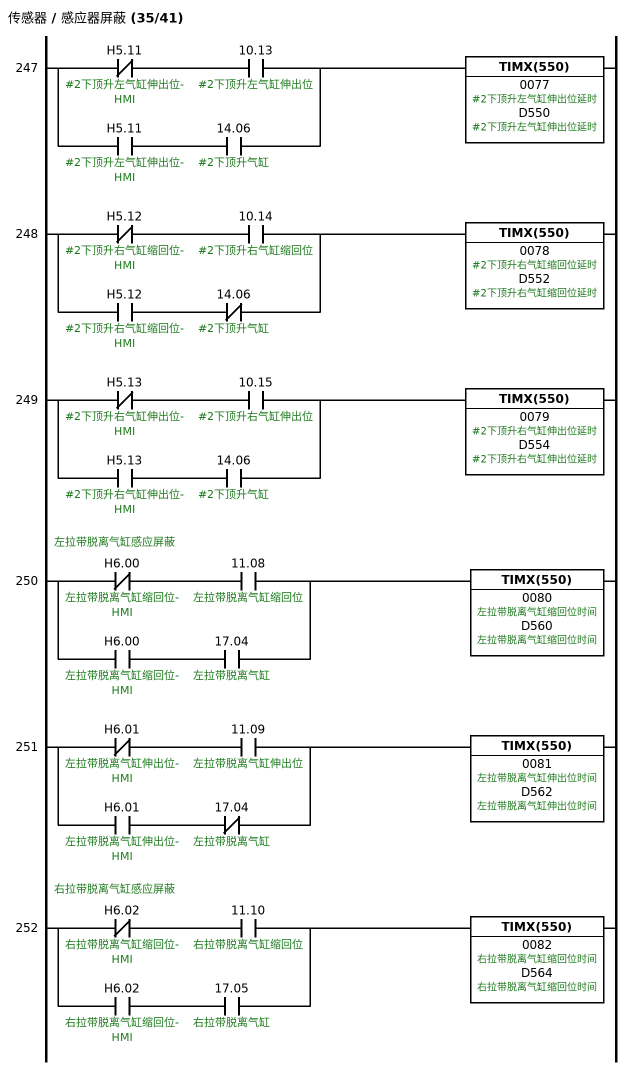
; rung 247
LDNOT H5.11  ; #2下顶升左气缸伸出位-HMI
AND 10.13  ; #2下顶升左气缸伸出位
LD H5.11  ; #2下顶升左气缸伸出位-HMI
AND 14.06  ; #2下顶升气缸
ORLD
TIMX(550) 0077 D550  ; #2下顶升左气缸伸出位延时
; rung 248
LDNOT H5.12  ; #2下顶升右气缸缩回位-HMI
AND 10.14  ; #2下顶升右气缸缩回位
LD H5.12  ; #2下顶升右气缸缩回位-HMI
ANDNOT 14.06  ; #2下顶升气缸
ORLD
TIMX(550) 0078 D552  ; #2下顶升右气缸缩回位延时
; rung 249
LDNOT H5.13  ; #2下顶升右气缸伸出位-HMI
AND 10.15  ; #2下顶升右气缸伸出位
LD H5.13  ; #2下顶升右气缸伸出位-HMI
AND 14.06  ; #2下顶升气缸
ORLD
TIMX(550) 0079 D554  ; #2下顶升右气缸伸出位延时
; rung 250: 左拉带脱离气缸感应屏蔽
LDNOT H6.00  ; 左拉带脱离气缸缩回位-HMI
AND 11.08  ; 左拉带脱离气缸缩回位
LD H6.00  ; 左拉带脱离气缸缩回位-HMI
AND 17.04  ; 左拉带脱离气缸
ORLD
TIMX(550) 0080 D560  ; 左拉带脱离气缸缩回位时间
; rung 251
LDNOT H6.01  ; 左拉带脱离气缸伸出位-HMI
AND 11.09  ; 左拉带脱离气缸伸出位
LD H6.01  ; 左拉带脱离气缸伸出位-HMI
ANDNOT 17.04  ; 左拉带脱离气缸
ORLD
TIMX(550) 0081 D562  ; 左拉带脱离气缸伸出位时间
; rung 252: 右拉带脱离气缸感应屏蔽
LDNOT H6.02  ; 右拉带脱离气缸缩回位-HMI
AND 11.10  ; 右拉带脱离气缸缩回位
LD H6.02  ; 右拉带脱离气缸缩回位-HMI
AND 17.05  ; 右拉带脱离气缸
ORLD
TIMX(550) 0082 D564  ; 右拉带脱离气缸缩回位时间

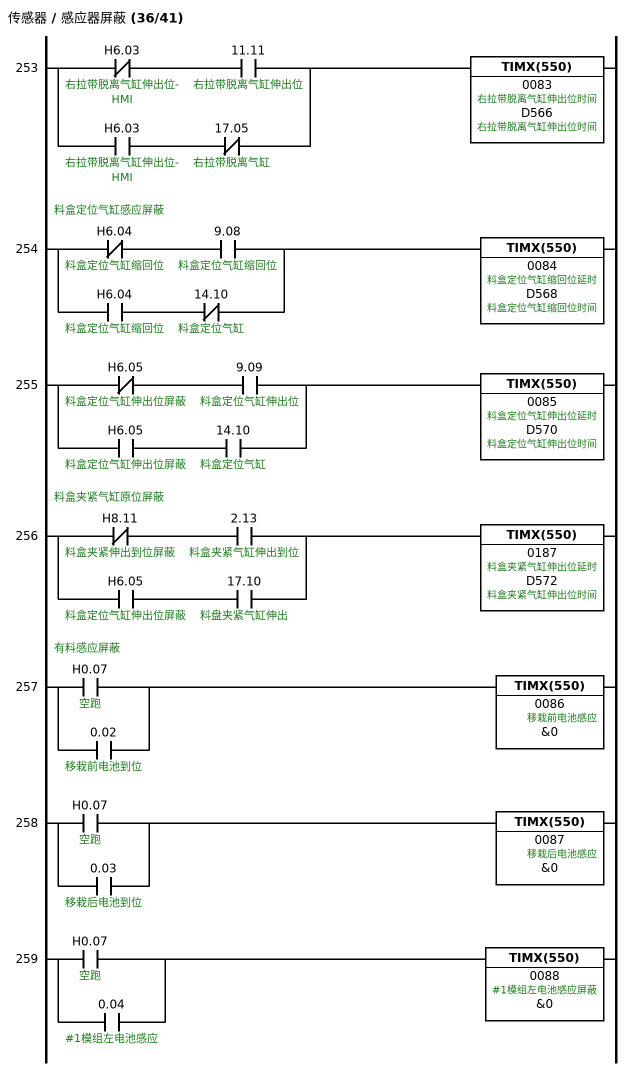
; rung 253
LDNOT H6.03  ; 右拉带脱离气缸伸出位-HMI
AND 11.11  ; 右拉带脱离气缸伸出位
LD H6.03  ; 右拉带脱离气缸伸出位-HMI
ANDNOT 17.05  ; 右拉带脱离气缸
ORLD
TIMX(550) 0083 D566  ; 右拉带脱离气缸伸出位时间
; rung 254: 料盒定位气缸感应屏蔽
LDNOT H6.04  ; 料盒定位气缸缩回位
AND 9.08  ; 料盒定位气缸缩回位
LD H6.04  ; 料盒定位气缸缩回位
ANDNOT 14.10  ; 料盒定位气缸
ORLD
TIMX(550) 0084 D568  ; 料盒定位气缸缩回位时间, 料盒定位气缸缩回位延时
; rung 255
LDNOT H6.05  ; 料盒定位气缸伸出位屏蔽
AND 9.09  ; 料盒定位气缸伸出位
LD H6.05  ; 料盒定位气缸伸出位屏蔽
AND 14.10  ; 料盒定位气缸
ORLD
TIMX(550) 0085 D570  ; 料盒定位气缸伸出位时间, 料盒定位气缸伸出位延时
; rung 256: 料盒夹紧气缸原位屏蔽
LDNOT H8.11  ; 料盒夹紧伸出到位屏蔽
AND 2.13  ; 料盒夹紧气缸伸出到位
LD H6.05  ; 料盒定位气缸伸出位屏蔽
AND 17.10  ; 料盘夹紧气缸伸出
ORLD
TIMX(550) 0187 D572  ; 料盒夹紧气缸伸出位时间, 料盒夹紧气缸伸出位延时
; rung 257: 有料感应屏蔽
LD H0.07  ; 空跑
OR 0.02  ; 移栽前电池到位
TIMX(550) 0086 &0  ; 移栽前电池感应
; rung 258
LD H0.07  ; 空跑
OR 0.03  ; 移栽后电池到位
TIMX(550) 0087 &0  ; 移栽后电池感应
; rung 259
LD H0.07  ; 空跑
OR 0.04  ; #1模组左电池感应
TIMX(550) 0088 &0  ; #1模组左电池感应屏蔽

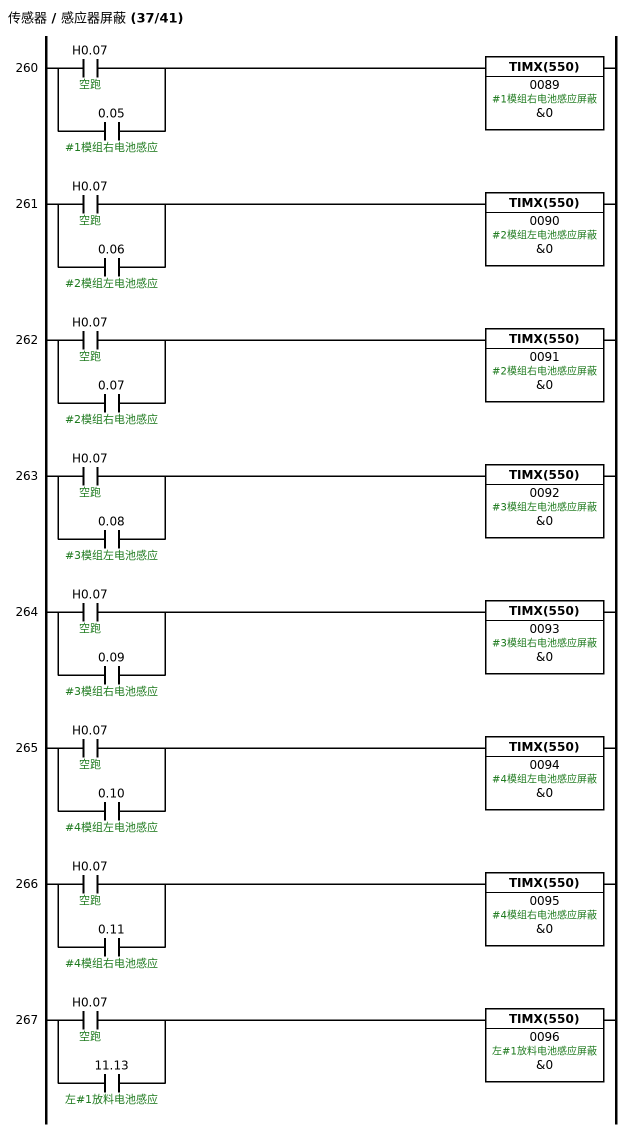
; rung 260
LD H0.07  ; 空跑
OR 0.05  ; #1模组右电池感应
TIMX(550) 0089 &0  ; #1模组右电池感应屏蔽
; rung 261
LD H0.07  ; 空跑
OR 0.06  ; #2模组左电池感应
TIMX(550) 0090 &0  ; #2模组左电池感应屏蔽
; rung 262
LD H0.07  ; 空跑
OR 0.07  ; #2模组右电池感应
TIMX(550) 0091 &0  ; #2模组右电池感应屏蔽
; rung 263
LD H0.07  ; 空跑
OR 0.08  ; #3模组左电池感应
TIMX(550) 0092 &0  ; #3模组左电池感应屏蔽
; rung 264
LD H0.07  ; 空跑
OR 0.09  ; #3模组右电池感应
TIMX(550) 0093 &0  ; #3模组右电池感应屏蔽
; rung 265
LD H0.07  ; 空跑
OR 0.10  ; #4模组左电池感应
TIMX(550) 0094 &0  ; #4模组左电池感应屏蔽
; rung 266
LD H0.07  ; 空跑
OR 0.11  ; #4模组右电池感应
TIMX(550) 0095 &0  ; #4模组右电池感应屏蔽
; rung 267
LD H0.07  ; 空跑
OR 11.13  ; 左#1放料电池感应
TIMX(550) 0096 &0  ; 左#1放料电池感应屏蔽

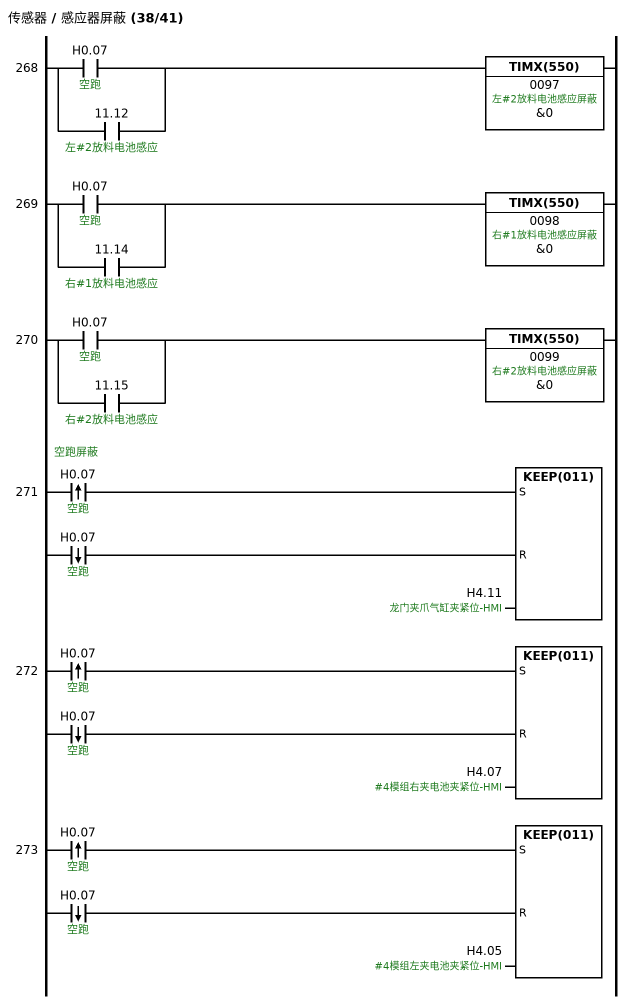
; rung 268
LD H0.07  ; 空跑
OR 11.12  ; 左#2放料电池感应
TIMX(550) 0097 &0  ; 左#2放料电池感应屏蔽
; rung 269
LD H0.07  ; 空跑
OR 11.14  ; 右#1放料电池感应
TIMX(550) 0098 &0  ; 右#1放料电池感应屏蔽
; rung 270
LD H0.07  ; 空跑
OR 11.15  ; 右#2放料电池感应
TIMX(550) 0099 &0  ; 右#2放料电池感应屏蔽
; rung 271: 空跑屏蔽
@LD H0.07  ; 空跑
%LD H0.07  ; 空跑
KEEP(011) H4.11  ; 龙门夹爪气缸夹紧位-HMI
; rung 272
@LD H0.07  ; 空跑
%LD H0.07  ; 空跑
KEEP(011) H4.07  ; #4模组右夹电池夹紧位-HMI
; rung 273
@LD H0.07  ; 空跑
%LD H0.07  ; 空跑
KEEP(011) H4.05  ; #4模组左夹电池夹紧位-HMI

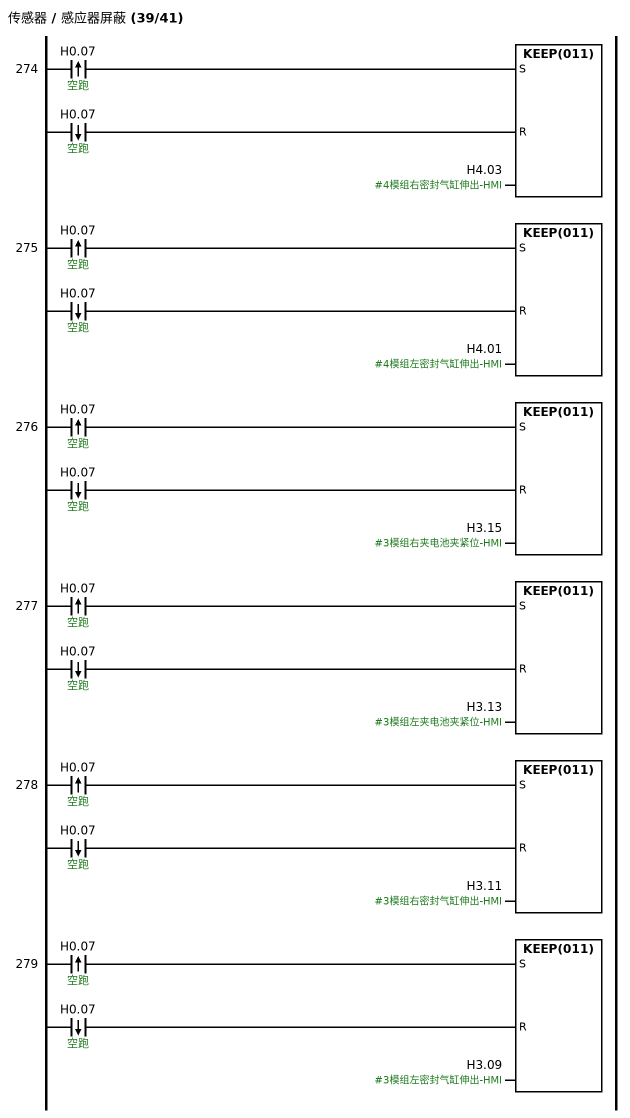
; rung 274
@LD H0.07  ; 空跑
%LD H0.07  ; 空跑
KEEP(011) H4.03  ; #4模组右密封气缸伸出-HMI
; rung 275
@LD H0.07  ; 空跑
%LD H0.07  ; 空跑
KEEP(011) H4.01  ; #4模组左密封气缸伸出-HMI
; rung 276
@LD H0.07  ; 空跑
%LD H0.07  ; 空跑
KEEP(011) H3.15  ; #3模组右夹电池夹紧位-HMI
; rung 277
@LD H0.07  ; 空跑
%LD H0.07  ; 空跑
KEEP(011) H3.13  ; #3模组左夹电池夹紧位-HMI
; rung 278
@LD H0.07  ; 空跑
%LD H0.07  ; 空跑
KEEP(011) H3.11  ; #3模组右密封气缸伸出-HMI
; rung 279
@LD H0.07  ; 空跑
%LD H0.07  ; 空跑
KEEP(011) H3.09  ; #3模组左密封气缸伸出-HMI

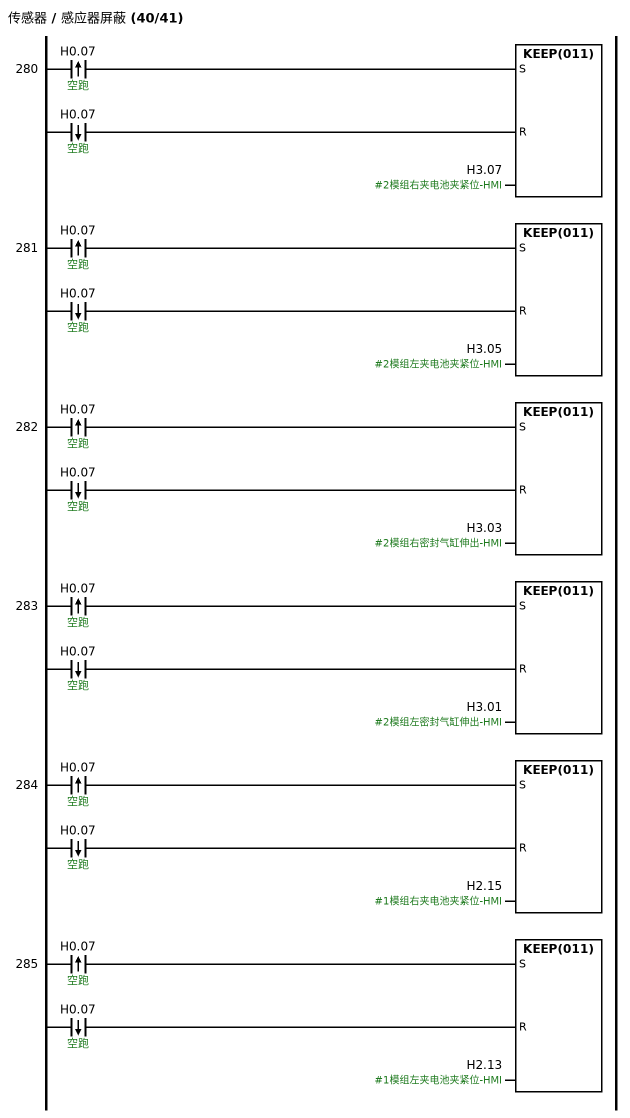
; rung 280
@LD H0.07  ; 空跑
%LD H0.07  ; 空跑
KEEP(011) H3.07  ; #2模组右夹电池夹紧位-HMI
; rung 281
@LD H0.07  ; 空跑
%LD H0.07  ; 空跑
KEEP(011) H3.05  ; #2模组左夹电池夹紧位-HMI
; rung 282
@LD H0.07  ; 空跑
%LD H0.07  ; 空跑
KEEP(011) H3.03  ; #2模组右密封气缸伸出-HMI
; rung 283
@LD H0.07  ; 空跑
%LD H0.07  ; 空跑
KEEP(011) H3.01  ; #2模组左密封气缸伸出-HMI
; rung 284
@LD H0.07  ; 空跑
%LD H0.07  ; 空跑
KEEP(011) H2.15  ; #1模组右夹电池夹紧位-HMI
; rung 285
@LD H0.07  ; 空跑
%LD H0.07  ; 空跑
KEEP(011) H2.13  ; #1模组左夹电池夹紧位-HMI

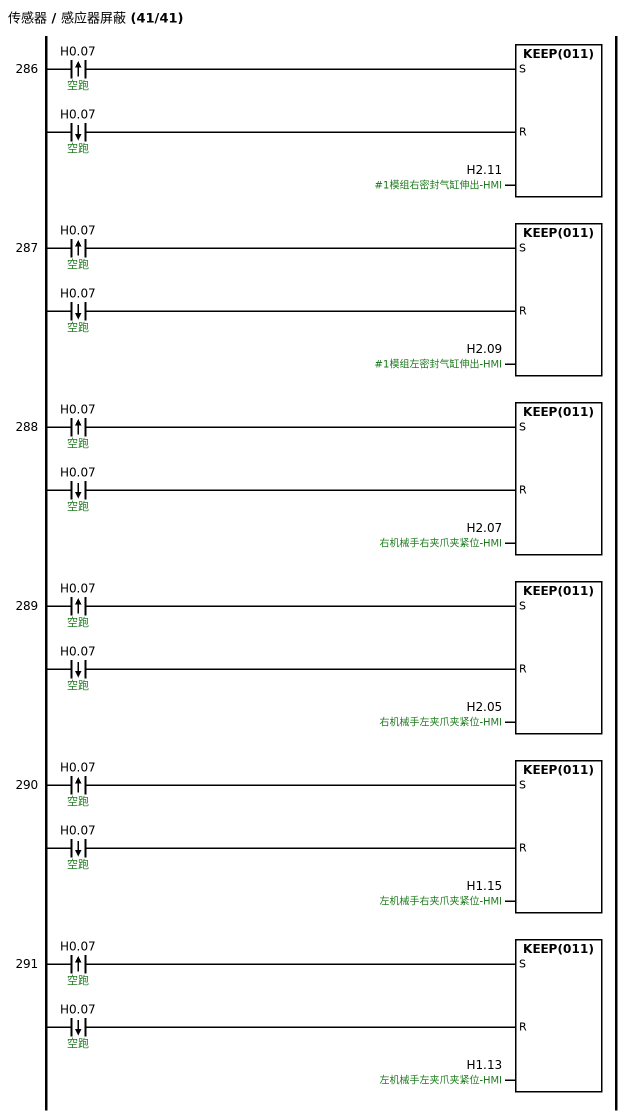
; rung 286
@LD H0.07  ; 空跑
%LD H0.07  ; 空跑
KEEP(011) H2.11  ; #1模组右密封气缸伸出-HMI
; rung 287
@LD H0.07  ; 空跑
%LD H0.07  ; 空跑
KEEP(011) H2.09  ; #1模组左密封气缸伸出-HMI
; rung 288
@LD H0.07  ; 空跑
%LD H0.07  ; 空跑
KEEP(011) H2.07  ; 右机械手右夹爪夹紧位-HMI
; rung 289
@LD H0.07  ; 空跑
%LD H0.07  ; 空跑
KEEP(011) H2.05  ; 右机械手左夹爪夹紧位-HMI
; rung 290
@LD H0.07  ; 空跑
%LD H0.07  ; 空跑
KEEP(011) H1.15  ; 左机械手右夹爪夹紧位-HMI
; rung 291
@LD H0.07  ; 空跑
%LD H0.07  ; 空跑
KEEP(011) H1.13  ; 左机械手左夹爪夹紧位-HMI

### Section 超时判断

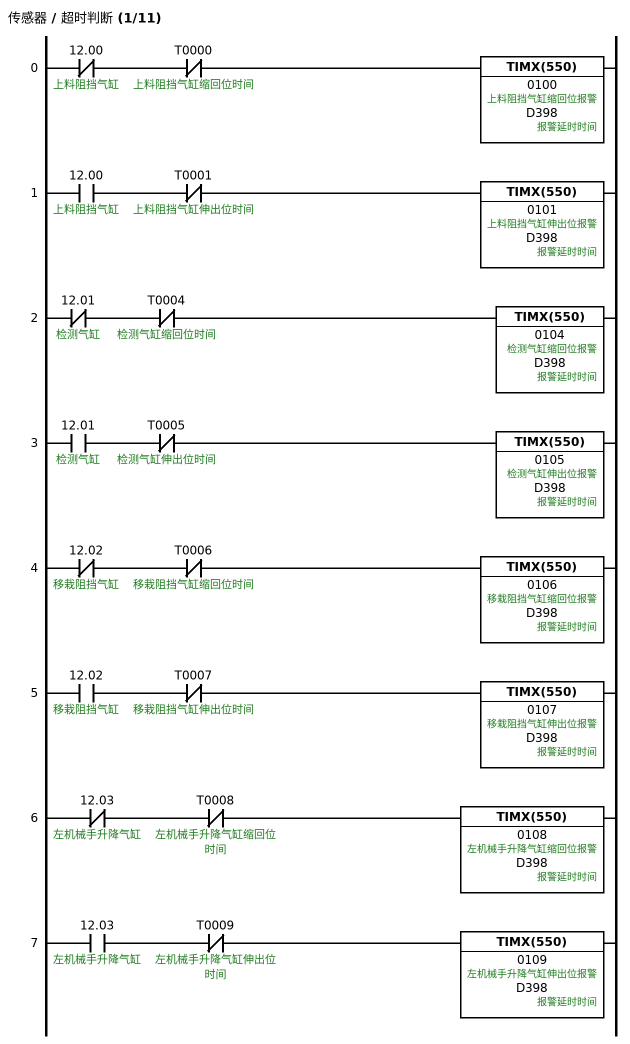
; rung 0
LDNOT 12.00  ; 上料阻挡气缸
ANDNOT T0000  ; 上料阻挡气缸缩回位时间
TIMX(550) 0100 D398  ; 报警延时时间, 上料阻挡气缸缩回位报警
; rung 1
LD 12.00  ; 上料阻挡气缸
ANDNOT T0001  ; 上料阻挡气缸伸出位时间
TIMX(550) 0101 D398  ; 报警延时时间, 上料阻挡气缸伸出位报警
; rung 2
LDNOT 12.01  ; 检测气缸
ANDNOT T0004  ; 检测气缸缩回位时间
TIMX(550) 0104 D398  ; 报警延时时间, 检测气缸缩回位报警
; rung 3
LD 12.01  ; 检测气缸
ANDNOT T0005  ; 检测气缸伸出位时间
TIMX(550) 0105 D398  ; 报警延时时间, 检测气缸伸出位报警
; rung 4
LDNOT 12.02  ; 移栽阻挡气缸
ANDNOT T0006  ; 移栽阻挡气缸缩回位时间
TIMX(550) 0106 D398  ; 报警延时时间, 移栽阻挡气缸缩回位报警
; rung 5
LD 12.02  ; 移栽阻挡气缸
ANDNOT T0007  ; 移栽阻挡气缸伸出位时间
TIMX(550) 0107 D398  ; 报警延时时间, 移栽阻挡气缸伸出位报警
; rung 6
LDNOT 12.03  ; 左机械手升降气缸
ANDNOT T0008  ; 左机械手升降气缸缩回位时间
TIMX(550) 0108 D398  ; 报警延时时间, 左机械手升降气缸缩回位报警
; rung 7
LD 12.03  ; 左机械手升降气缸
ANDNOT T0009  ; 左机械手升降气缸伸出位时间
TIMX(550) 0109 D398  ; 报警延时时间, 左机械手升降气缸伸出位报警

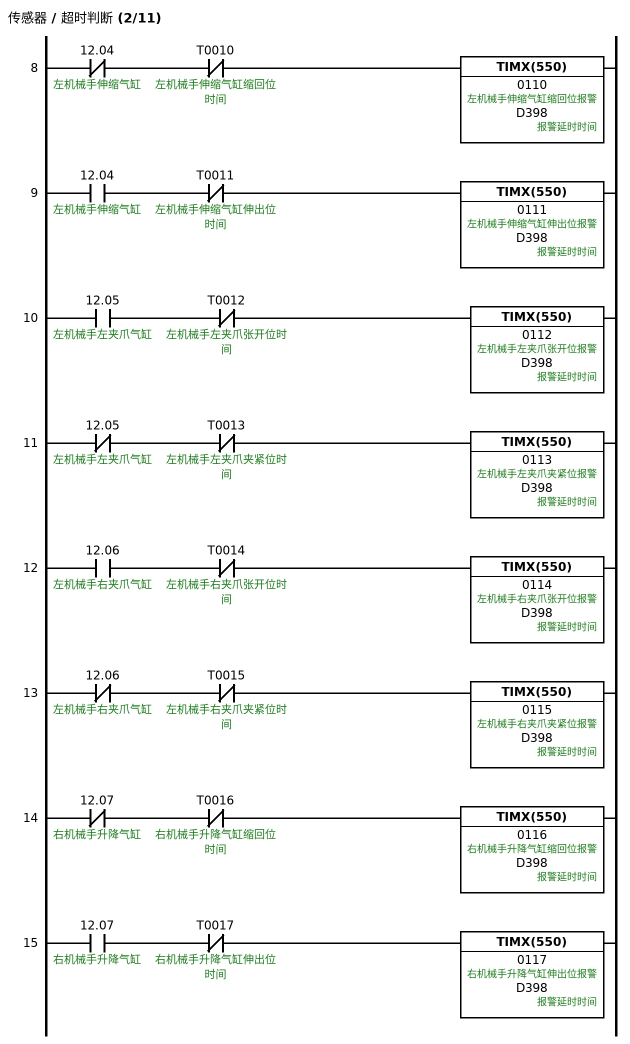
; rung 8
LDNOT 12.04  ; 左机械手伸缩气缸
ANDNOT T0010  ; 左机械手伸缩气缸缩回位时间
TIMX(550) 0110 D398  ; 报警延时时间, 左机械手伸缩气缸缩回位报警
; rung 9
LD 12.04  ; 左机械手伸缩气缸
ANDNOT T0011  ; 左机械手伸缩气缸伸出位时间
TIMX(550) 0111 D398  ; 报警延时时间, 左机械手伸缩气缸伸出位报警
; rung 10
LD 12.05  ; 左机械手左夹爪气缸
ANDNOT T0012  ; 左机械手左夹爪张开位时间
TIMX(550) 0112 D398  ; 报警延时时间, 左机械手左夹爪张开位报警
; rung 11
LDNOT 12.05  ; 左机械手左夹爪气缸
ANDNOT T0013  ; 左机械手左夹爪夹紧位时间
TIMX(550) 0113 D398  ; 报警延时时间, 左机械手左夹爪夹紧位报警
; rung 12
LD 12.06  ; 左机械手右夹爪气缸
ANDNOT T0014  ; 左机械手右夹爪张开位时间
TIMX(550) 0114 D398  ; 报警延时时间, 左机械手右夹爪张开位报警
; rung 13
LDNOT 12.06  ; 左机械手右夹爪气缸
ANDNOT T0015  ; 左机械手右夹爪夹紧位时间
TIMX(550) 0115 D398  ; 报警延时时间, 左机械手右夹爪夹紧位报警
; rung 14
LDNOT 12.07  ; 右机械手升降气缸
ANDNOT T0016  ; 右机械手升降气缸缩回位时间
TIMX(550) 0116 D398  ; 报警延时时间, 右机械手升降气缸缩回位报警
; rung 15
LD 12.07  ; 右机械手升降气缸
ANDNOT T0017  ; 右机械手升降气缸伸出位时间
TIMX(550) 0117 D398  ; 报警延时时间, 右机械手升降气缸伸出位报警

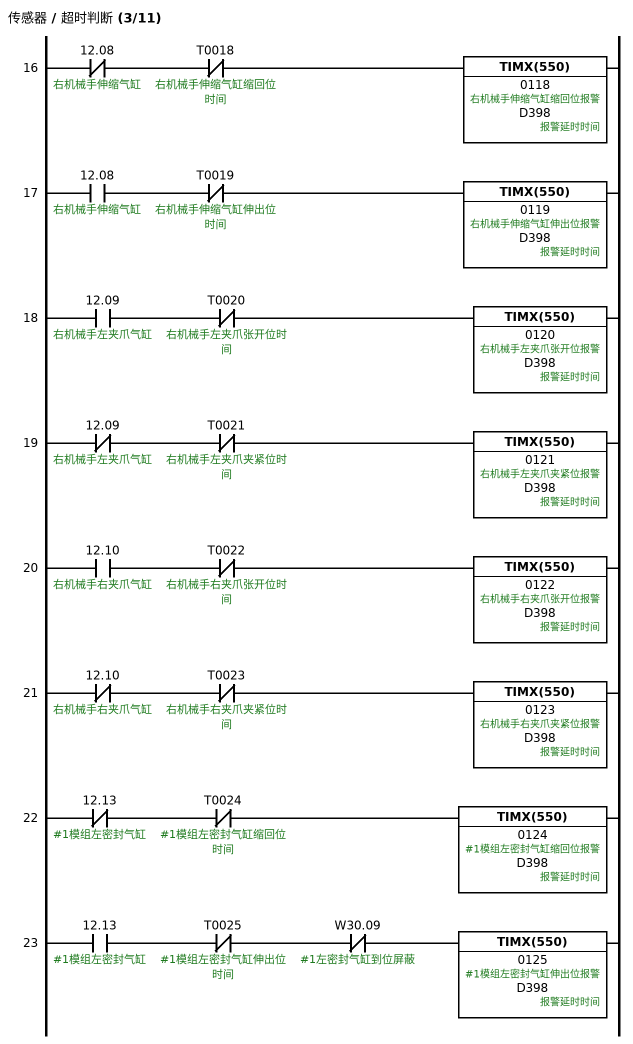
; rung 16
LDNOT 12.08  ; 右机械手伸缩气缸
ANDNOT T0018  ; 右机械手伸缩气缸缩回位时间
TIMX(550) 0118 D398  ; 报警延时时间, 右机械手伸缩气缸缩回位报警
; rung 17
LD 12.08  ; 右机械手伸缩气缸
ANDNOT T0019  ; 右机械手伸缩气缸伸出位时间
TIMX(550) 0119 D398  ; 报警延时时间, 右机械手伸缩气缸伸出位报警
; rung 18
LD 12.09  ; 右机械手左夹爪气缸
ANDNOT T0020  ; 右机械手左夹爪张开位时间
TIMX(550) 0120 D398  ; 报警延时时间, 右机械手左夹爪张开位报警
; rung 19
LDNOT 12.09  ; 右机械手左夹爪气缸
ANDNOT T0021  ; 右机械手左夹爪夹紧位时间
TIMX(550) 0121 D398  ; 报警延时时间, 右机械手左夹爪夹紧位报警
; rung 20
LD 12.10  ; 右机械手右夹爪气缸
ANDNOT T0022  ; 右机械手右夹爪张开位时间
TIMX(550) 0122 D398  ; 报警延时时间, 右机械手右夹爪张开位报警
; rung 21
LDNOT 12.10  ; 右机械手右夹爪气缸
ANDNOT T0023  ; 右机械手右夹爪夹紧位时间
TIMX(550) 0123 D398  ; 报警延时时间, 右机械手右夹爪夹紧位报警
; rung 22
LDNOT 12.13  ; #1模组左密封气缸
ANDNOT T0024  ; #1模组左密封气缸缩回位时间
TIMX(550) 0124 D398  ; 报警延时时间, #1模组左密封气缸缩回位报警
; rung 23
LD 12.13  ; #1模组左密封气缸
ANDNOT T0025  ; #1模组左密封气缸伸出位时间
ANDNOT W30.09  ; #1左密封气缸到位屏蔽
TIMX(550) 0125 D398  ; 报警延时时间, #1模组左密封气缸伸出位报警

